// TIA Portal V20 export
TYPE "LPFE_typeStatus"
// stored: Access Published, Namespace PFE
   STRUCT
      Maintenance : Struct
         MS : Struct
            "kDiag.Alarm.MaintStatusPLCForceEdit" : Int := 251;   // PLC Forces and/or Edits Present and/or Active
            "kDiag.Alarm.MaintStatusGeneral" : Int := 254;   // Maintenance Status General
         END_STRUCT;
      END_STRUCT;
      Production : Struct
         PS : Struct
            "kDiag.Alarm.ProdStatus" : Int := 255;   // Production Status
            "kDiag.Alarm.ProdStatusAndon" : Int := 256;
         END_STRUCT;
      END_STRUCT;
      Tooling : Struct
         LS : Struct
            "kDiag.Alarm.ToolStatus" : Int := 260;   // Tooling Status
         END_STRUCT;
      END_STRUCT;
      Quality : Struct
         QS : Struct
            "kDiag.Alarm.QualStatus" : Int := 265;   // Quality Status
         END_STRUCT;
      END_STRUCT;
      Throughput : Struct
         TS : Struct
            "kDiag.Alarm.TputStatus" : Int := 270;   // Thruput Status
         END_STRUCT;
      END_STRUCT;
      System : Struct
         SS : Struct
            "kDiag.Alarm.SysStatus" : Int := 275;   // System Status
         END_STRUCT;
      END_STRUCT;
      Material : Struct
         AS : Struct
            "kDiag.Alarm.MatlStatus" : Int := 280;   // Material Status
         END_STRUCT;
      END_STRUCT;
   END_STRUCT;
END_TYPE
